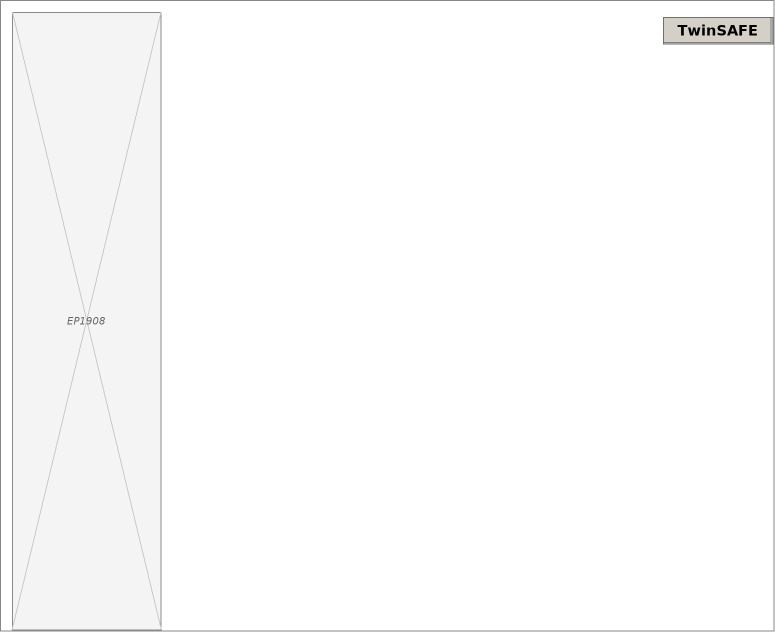
VISUALIZATION EP1908_Specific_Diagnostics  // 775x632
    Button (663,17 110x27), "TwinSAFE"
        OnMouseClick: change screen: TwinSAFE
        OnMouseUp: execute { g_xHMI_ErrAckPB := FALSE ; }
    Image (12,12 149x618), image: EP1908
END_VISUALIZATION

(* stored: Version 1.1.0.1, ProductVersion 3.1.0.18
   Visu EP1908_Specific_Diagnostics: Id {5aa348b4-08bf-47a0-88e9-a3aa05c9958c} *)
